# EPICS substitutions: pnan5221/Db/pnan5221.substitutions
file "pnan5221-gen.template" { pattern {}
{}
}

file "pnan5221-trace.template" { pattern
{N, MTRNR}
{1  1}
{2  1}
{3  2}
}
